// TIA Portal V20 export
TYPE "typeSequenceControlNodeJobInterface_sideTapeLoading"
// stored: Namespace Unit1.Em4
   STRUCT
      chargeJob2 : "LER_typeJobInterface";
   END_STRUCT;
END_TYPE
